{attribute 'GeneratedUsingTerminal: KL2791'}
{attribute addProperty BoxType "KL2791"}
{attribute addProperty Id "Channel_1AT %Q*Channel_6576A6810"}
{attribute addProperty CRC "1632160004"}
{attribute addProperty Size "0"}
TYPE KL2791_6148C904 :
STRUCT
	{attribute addProperty Name "Channel_1"}
	Channel_1 : Channel_6576A681;
END_STRUCT
END_TYPE

(* stored: Version 1.2.0.0, ProductVersion 3.1.4024.9
   DUT KL2791_6148C904: Id {4adc83d8-9f9b-4f70-9f56-cb437665f50a} *)
